// Mitsubishi GX Works2 project: counter   PLC: Q03UDV

PROGRAM MAIN
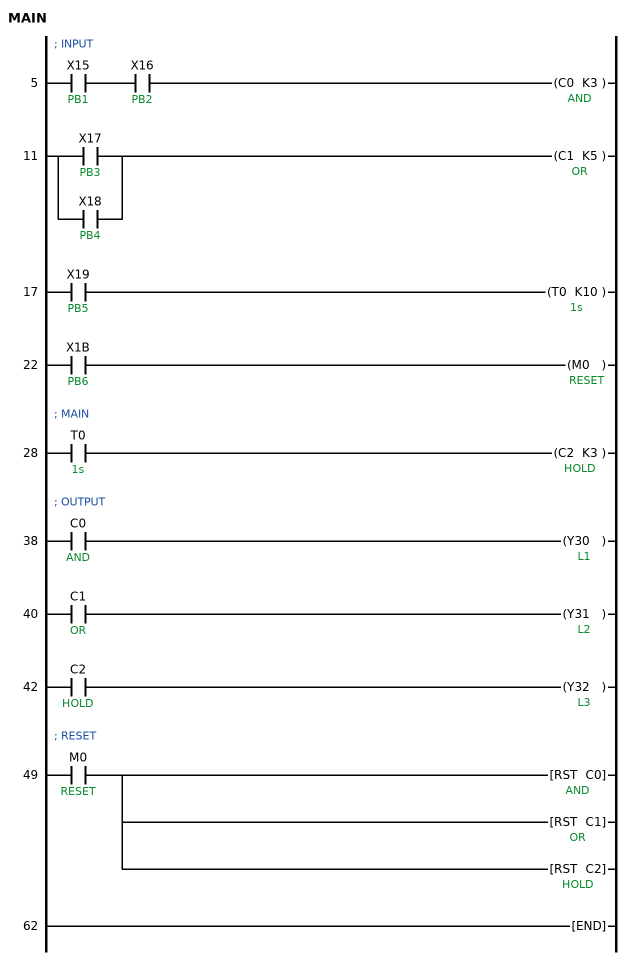
; INPUT
5     LD      X15  ; PB1
      AND     X16  ; PB2
      OUT     C0 K3  ; AND
11    LD      X17  ; PB3
      OR      X18  ; PB4
      OUT     C1 K5  ; OR
17    LD      X19  ; PB5
      OUT     T0 K10  ; 1s
22    LD      X1B  ; PB6
      OUT     M0  ; RESET
; MAIN
28    LD      T0  ; 1s
      OUT     C2 K3  ; HOLD
; OUTPUT
38    LD      C0  ; AND
      OUT     Y30  ; L1
40    LD      C1  ; OR
      OUT     Y31  ; L2
42    LD      C2  ; HOLD
      OUT     Y32  ; L3
; RESET
49    LD      M0  ; RESET
      RST     C0  ; AND
      RST     C1  ; OR
      RST     C2  ; HOLD
62    END
END_PROGRAM
